{attribute 'qualified_only'}
{attribute 'strict'}
TYPE E_SafetyStates :
(
	IDLE := 0,
	CHECK_SAFETY_INPUTS,
	CHECK_DOOR_CLOSED,
	CHECK_DOOR_LOCKED,
	LOCKDOOR_REQUEST,
	CHECK_DOOR_OSSD,
	CHECK_SAFETY_OUTPUT,
	DOOR_LOCK,
	TRIG_RESET,
	CHECK_OTHER_STATION,
	DONE,
	ERROR
);
END_TYPE

(* stored: Version 1.1.0.1, ProductVersion 3.1.4024.12
   DUT E_SafetyStates: Id {19627ce2-aab1-4347-990c-5641411672d1} *)
